KUKA KRL program: pickbox1.src, pickbox1.dat

--- pickbox1.src ---
&ACCESS RVO1
&COMMENT
&ACCESS RVO
&PARAM EDITMASK = *
&PARAM TEMPLATE = C:\KRC\Roboter\Template\vorgabe
&PARAM DISKPATH = KRC:\R1\Program\program_1
DEF pickbox1(X_box:in)
DECL POS X_box

XP1.x = XP1m.x + 3 * (395 - X_box)
XP2.x = XP1.x
XP3.x = XP1.x
XP4.x = XP1.x
XP5.x = XP1.x

;FOLD PTP HOME  Vel=100 % DEFAULT Tool[2]:tool_empty Base[0];%{PE}%R 8.3.22,%MKUKATPBASIS,%CMOVE,%VPTP,%P 1:PTP, 2:HOME, 3:, 5:100, 7:DEFAULT
$BWDSTART=FALSE
PDAT_ACT=PDEFAULT
FDAT_ACT=FHOME
BAS(#PTP_PARAMS,100)
PTP XHOME
;ENDFOLD

IF (Air_Supply_OK == FALSE) THEN
    HALT
    $MSG_T.TYP = #quit
    $MSG_T.KEY[]="Davleniye vozdukha ne v norme" ;MSG
    $MSG_T.VALID=TRUE ;vivvod MSG
    ; wait for aknowledgement
    WHILE  $MSG_T.VALID == true
    ; WAIT SEC 0.05
    ENDWHILE
ENDIF

; approach
;FOLD LIN P1 CONT Vel=2.00000 m/s CPDAT1 Tool[2]:tool_empty Base[3]:pickbox1;%{PE}%R 8.3.22,%MKUKATPBASIS,%CMOVE,%VLIN,%P 1:LIN, 2:P1, 3:C_DIS C_DIS, 5:2.00000, 7:CPDAT1
$BWDSTART=FALSE
LDAT_ACT=LCPDAT1
FDAT_ACT=FP1
BAS(#CP_PARAMS,2.00000)
LIN XP1 C_DIS C_DIS
;ENDFOLD

; descent to wall
;FOLD LIN P2 CONT Vel=2.00000 m/s CPDAT2 Tool[2]:tool_empty Base[3]:pickbox1;%{PE}%R 8.3.22,%MKUKATPBASIS,%CMOVE,%VLIN,%P 1:LIN, 2:P2, 3:C_DIS C_DIS, 5:2.00000, 7:CPDAT2
$BWDSTART=FALSE
LDAT_ACT=LCPDAT2
FDAT_ACT=FP2
BAS(#CP_PARAMS,2.00000)
LIN XP2 C_DIS C_DIS
;ENDFOLD

;moving boxes from the wall
;FOLD LIN P3 CONT Vel=2.00000 m/s CPDAT3 Tool[3]:tool_2_box Base[3]:pickbox1;%{PE}%R 8.3.22,%MKUKATPBASIS,%CMOVE,%VLIN,%P 1:LIN, 2:P3, 3:C_DIS C_DIS, 5:2.00000, 7:CPDAT3
$BWDSTART=FALSE
LDAT_ACT=LCPDAT3
FDAT_ACT=FP3
BAS(#CP_PARAMS,2.00000)
LIN XP3 C_DIS C_DIS
;ENDFOLD

; descent
;FOLD LIN P4 CONT Vel=2.00000 m/s CPDAT4 Tool[2]:tool_empty Base[3]:pickbox1;%{PE}%R 8.3.22,%MKUKATPBASIS,%CMOVE,%VLIN,%P 1:LIN, 2:P4, 3:C_DIS C_DIS, 5:2.00000, 7:CPDAT4
$BWDSTART=FALSE
LDAT_ACT=LCPDAT4
FDAT_ACT=FP4
BAS(#CP_PARAMS,2.00000)
LIN XP4 C_DIS C_DIS
;ENDFOLD

; pick up boxes
;FOLD OUT 1 'finger right'  State= TRUE;%{PE}%R 8.3.22,%MKUKATPBASIS,%COUT,%VOUTX,%P 2:1, 3:finger right, 5:TRUE, 6:

$OUT[1]=TRUE
;ENDFOLD
;FOLD OUT 3 'finger left'  State= TRUE;%{PE}%R 8.3.22,%MKUKATPBASIS,%COUT,%VOUTX,%P 2:3, 3:finger left, 5:TRUE, 6:

$OUT[3]=TRUE
;ENDFOLD
;FOLD WAIT Time= 0.5 sec;%{PE}%R 8.3.22,%MKUKATPBASIS,%CWAIT,%VWAIT,%P 2:0.5
WAIT SEC 0.5
;ENDFOLD

; pulling out the support
;FOLD OUT 2 'support hook right' State=TRUE ;%{PE}%R 8.3.32,%MKUKATPBASIS,%COUT,%VOUTX,%P 2:2, 3:support hook right, 5:TRUE, 6:
$OUT[2]=TRUE
;ENDFOLD
;FOLD OUT 4 'support hook left' State=TRUE ;%{PE}%R 8.3.32,%MKUKATPBASIS,%COUT,%VOUTX,%P 2:4, 3:support hook left, 5:TRUE, 6:
$OUT[4]=TRUE
;ENDFOLD
;FOLD WAIT Time=1 sec;%{PE}%R 8.3.32,%MKUKATPBASIS,%CWAIT,%VWAIT,%P 3:1
WAIT SEC 1
;ENDFOLD

L1_Product_Picked = TRUE

; taking boxes out
;FOLD LIN P5  Vel=2.00000 m/s CPDAT5 Tool[3]:tool_2_box Base[3]:pickbox1;%{PE}%R 8.3.22,%MKUKATPBASIS,%CMOVE,%VLIN,%P 1:LIN, 2:P5, 3:, 5:2.00000, 7:CPDAT5
$BWDSTART=FALSE
LDAT_ACT=LCPDAT5
FDAT_ACT=FP5
BAS(#CP_PARAMS,2.00000)
LIN XP5
;ENDFOLD

;check for allowance to leave the pick point zone
IF (L1_Pick_Point_Clear == FALSE) THEN
    $MSG_T.TYP = #quit
    $MSG_T.KEY[]="Net razresheniya pokinut' zonu vzyatiya korobok" ;MSG
    $MSG_T.VALID=TRUE ;vivvod MSG
    ; wait for aknowledgement
    WHILE  $MSG_T.VALID == true
    ; WAIT SEC 0.05
    ENDWHILE
ENDIF
;FOLD WAIT FOR ( L1_Pick_Point_Clear  );%{PE}%R 8.3.22,%MKUKATPBASIS,%CEXT_WAIT_FOR,%VEXT_WAIT_FOR,%P 2:, 4:, 5:L1_Pick_Point_Clear, 6:1, 7:, 9:
WAIT FOR  (  (L1_Pick_Point_Clear) )
;ENDFOLD

L1_Product_Picked = FALSE ; reset the signal

; depature
;FOLD LIN P6 CONT Vel=2.00000 m/s CPDAT1 Tool[3]:tool_2_box Base[3]:pickbox1;%{PE}%R 8.3.22,%MKUKATPBASIS,%CMOVE,%VLIN,%P 1:LIN, 2:P6, 3:C_DIS C_DIS, 5:2.00000, 7:CPDAT1
$BWDSTART=FALSE
LDAT_ACT=LCPDAT6
FDAT_ACT=FP6
BAS(#CP_PARAMS,2.00000)
LIN XP6 C_DIS C_DIS
;ENDFOLD

; movement to home
;FOLD PTP HOME  Vel= 100 % DEFAULT;%{PE}%MKUKATPBASIS,%CMOVE,%VPTP,%P 1:PTP, 2:HOME, 3:, 5:100, 7:DEFAULT
$BWDSTART = FALSE
PDAT_ACT=PDEFAULT
FDAT_ACT=FHOME
BAS (#PTP_PARAMS,100 )
$H_POS=XHOME
PTP  XHOME
;ENDFOLD

END

--- pickbox1.dat ---
&ACCESS RVO1
&COMMENT
DEFDAT pickbox1 PUBLIC
;FOLD EXTERNAL DECLARATIONS;%{PE}%MKUKATPBASIS,%CEXT,%VCOMMON,%P
;FOLD BASISTECH EXT;%{PE}%MKUKATPBASIS,%CEXT,%VEXT,%P
EXT  BAS (BAS_COMMAND  :IN,REAL  :IN )
DECL INT SUCCESS
;ENDFOLD (BASISTECH EXT)
;FOLD USER EXT;%{E}%MKUKATPUSER,%CEXT,%VEXT,%P
;Make here your modifications

;ENDFOLD (USER EXT)
;ENDFOLD (EXTERNAL DECLERATIONS)
; DECL BASIS_SUGG_T LAST_BASIS={POINT1[] "P5                    ",POINT2[] "P5                    ",CP_PARAMS[] "CPDAT5                 ",PTP_PARAMS[] "PDAT1                   ",CONT[] "C_DIS C_DIS             ",CP_VEL[] "0.1                     ",PTP_VEL[] "20                      ",SYNC_PARAMS[] "SYNCDAT                 ",SPL_NAME[] "S0                      ",A_PARAMS[] "ADAT0                   "}
DECL PDAT PPDAT1={VEL 100.000,ACC 100.000,APO_DIST 100.000,APO_MODE #CDIS,GEAR_JERK 50.0000}
DECL E6POS XP1={X 1463.90698,Y -2335.81665,Z 678.544678,A 1.96151149,B -8.27161622E-14,C -180.000,S 2,T 3,E1 0.0,E2 0.0,E3 0.0,E4 0.0,E5 0.0,E6 0.0}
DECL FDAT FP1={TOOL_NO 2,BASE_NO 3,IPO_FRAME #BASE,POINT2[] " ",TQ_STATE FALSE}
DECL LDAT LCPDAT1={VEL 2.00000,ACC 100,APO_DIST 100,APO_FAC 50,AXIS_VEL 100.0,AXIS_ACC 100.0,ORI_TYP #VAR,CIRC_TYP #BASE,JERK_FAC 50.0,GEAR_JERK 50.0,EXAX_IGN 0}
DECL E6POS XP2={X 1463.90674,Y -2335.81665,Z 609.857727,A 1.96151149,B 3.12117546E-13,C 180.000,S 2,T 3,E1 0.0,E2 0.0,E3 0.0,E4 0.0,E5 0.0,E6 0.0}
DECL FDAT FP2={TOOL_NO 2,BASE_NO 3,IPO_FRAME #BASE,POINT2[] " ",TQ_STATE FALSE}
DECL LDAT LCPDAT2={VEL 2.00000,ACC 100,APO_DIST 100,APO_FAC 50,AXIS_VEL 100.0,AXIS_ACC 100.0,ORI_TYP #VAR,CIRC_TYP #BASE,JERK_FAC 50.0,GEAR_JERK 50.0,EXAX_IGN 0}
DECL E6POS XP3={X 1463.90527,Y -2335.81689,Z 428.891693,A 1.96151149,B -4.43258745E-14,C -180.000,S 2,T 3,E1 0.0,E2 0.0,E3 0.0,E4 0.0,E5 0.0,E6 0.0}
DECL FDAT FP3={TOOL_NO 3,BASE_NO 3,IPO_FRAME #BASE,POINT2[] " ",TQ_STATE FALSE}
DECL LDAT LCPDAT3={VEL 2.00000,ACC 100,APO_DIST 100,APO_FAC 50,AXIS_VEL 100.0,AXIS_ACC 100.0,ORI_TYP #VAR,CIRC_TYP #BASE,JERK_FAC 50.0,GEAR_JERK 50.0,EXAX_IGN 0}
DECL E6POS XP4={X 1463.90527,Y -2321.53149,Z 428.891693,A 1.96151149,B -2.25146931E-14,C -180.000,S 2,T 3,E1 0.0,E2 0.0,E3 0.0,E4 0.0,E5 0.0,E6 0.0}
DECL FDAT FP4={TOOL_NO 2,BASE_NO 3,IPO_FRAME #BASE,POINT2[] " ",TQ_STATE FALSE}
DECL LDAT LCPDAT4={VEL 2.00000,ACC 100,APO_DIST 100,APO_FAC 50,AXIS_VEL 100.0,AXIS_ACC 100.0,ORI_TYP #VAR,CIRC_TYP #BASE,JERK_FAC 50.0,GEAR_JERK 50.0,EXAX_IGN 0}
DECL E6POS XP5={X 1463.90527,Y -1124.04126,Z 456.946777,A 1.95980179,B -9.74044860E-15,C -180.000,S 2,T 3,E1 0.0,E2 0.0,E3 0.0,E4 0.0,E5 0.0,E6 0.0}
DECL FDAT FP5={TOOL_NO 3,BASE_NO 3,IPO_FRAME #BASE,POINT2[] " ",TQ_STATE FALSE}
DECL LDAT LCPDAT5={VEL 2.00000,ACC 100,APO_DIST 100,APO_FAC 50,AXIS_VEL 100.0,AXIS_ACC 100.0,ORI_TYP #VAR,CIRC_TYP #BASE,JERK_FAC 50.0,GEAR_JERK 50.0,EXAX_IGN 0}
DECL E6POS XP6={X 1463.90698,Y -2335.81665,Z 678.544678,A 1.96151149,B -8.27161622E-14,C -180.000,S 2,T 3,E1 0.0,E2 0.0,E3 0.0,E4 0.0,E5 0.0,E6 0.0}
DECL FDAT FP6={TOOL_NO 3,BASE_NO 3,IPO_FRAME #BASE,POINT2[] " ",TQ_STATE FALSE}
DECL LDAT LCPDAT6={VEL 2.00000,ACC 100,APO_DIST 100,APO_FAC 50,AXIS_VEL 100.0,AXIS_ACC 100.0,ORI_TYP #VAR,CIRC_TYP #BASE,JERK_FAC 50.0,GEAR_JERK 50.0,EXAX_IGN 0}
DECL E6POS XP1m={X 1463.90698,Y -2335.81665,Z 678.544678,A 1.96151149,B -8.27161622E-14,C -180.000,S 2,T 3,E1 0.0,E2 0.0,E3 0.0,E4 0.0,E5 0.0,E6 0.0}
DECL FDAT FP1m={TOOL_NO 2,BASE_NO 3,IPO_FRAME #BASE,POINT2[] " ",TQ_STATE FALSE}
ENDDAT
